// TwinCAT 3 PLC project ForgeExample
// ProgramVersion: 3.1.4026.17
// libraries:
//   Tc2_Standard, * (Beckhoff Automation GmbH)
//   Tc2_System, * (Beckhoff Automation GmbH)
//   Tc3_JsonXml, * (Beckhoff Automation GmbH)
//   Tc3_Module, * (Beckhoff Automation GmbH)
//   [Twincat Open Library], * (Home)
//   VisuSymbols,3.5.10.0,System
// project tree:
//   DUTs/ ST_CameraStates.TcDUT (not stored)
//   GVLs/ Hardware_Mapping.TcGVL (not stored), Cognex_Mapping.TcGVL (not stored)
//   / PlcTask.TcTTO
//   POUs/ MAIN.TcPOU, _5000_PRG_Aborting.TcPOU (not stored), _1000_PRG_Homing.TcPOU, _3000_PRG_Running.TcPOU (not stored), _2000_PRG_Stopping.TcPOU (not stored), _4000_PRG_Pausing.TcPOU (not stored), _6000_PRG_Proceeding.TcPOU (not stored)
// real-time tasks:
//   TASK PlcTask: cycle T#10ms, priority 20, ADS port 350
//   TASK VISU_TASK: cycle T#200000us, priority 30, ADS port 351
//   TASK IO Task New: cycle T#1ms, priority 1, ADS port 301
// motion (NC):
//   TASK NC-Task 1 SAF: cycle T#2ms, priority 4, ADS port 501
//   TASK NC-Task 1 SVB: cycle T#10ms, priority 8, ADS port 511
//   AXIS Axis 1 (id 1)
//     OtherSettings: AllowMotionCmdToSlave=true
//     encoder EncType=4
//       EncPara: MaxCount=#x0000ffff
//         Inc: RefSoftSyncMask=#x0000ffff
//     drive DrvType=24
//       Analog: TorqueSetpointScale=10, ScaleFactorActTorque=0.1
//       TimeComp: TaskDelayCycles=1
//     controller CtrType=1
//       CtrPara: PriorControlFactor=1
//         Observer: BandWidth=20
//   AXIS Axis 2 (id 2)
//     OtherSettings: AllowMotionCmdToSlave=true
//     encoder EncType=4
//       EncPara: MaxCount=#x0000ffff
//         Inc: RefSoftSyncMask=#x0000ffff
//     drive DrvType=24
//       Analog: TorqueSetpointScale=10, ScaleFactorActTorque=0.1
//       TimeComp: TaskDelayCycles=1
//     controller CtrType=1
//       CtrPara: PriorControlFactor=1
//         Observer: BandWidth=20
// I/O:
//   DEVICE Device 1 (TC3 EIP Scanner), AmsNetId 172.18.236.100.2.1
//     Box 1 (In-Sight 7000 Series) // <INFO> </INFO> <EDS> C:\TwinCAT\3.1\Config\Io\EtherNetIP\02A6006401090C00.eds </EDS>
//   DEVICE Device 2 (EtherCAT), AmsNetId 172.18.236.100.3.1
//     Term 2 (EK1100) [EK1100 EtherCAT Coupler (2A E-Bus)]
//       Term 3 (EL1008) [EL1008 8Ch. Dig. Input 24V, 3ms]
//       Term 4 (EL1008) [EL1008 8Ch. Dig. Input 24V, 3ms]
//       Term 5 (EL2008) [EL2008 8Ch. Dig. Output 24V, 0.5A]
//       Term 6 (EL2008) [EL2008 8Ch. Dig. Output 24V, 0.5A]
//       Term 7 (EL7047) [EL7047 1Ch. Stepper motor output stage (50V, 5A)]
//       Term 8 (EL7047) [EL7047 1Ch. Stepper motor output stage (50V, 5A)]
//       Term 8 (EL9011) [EL9011 End Terminal]
// variable links:
//   NC-Task 1 SAF/Axes/Axis 1 <-> Device 2 (EtherCAT)/Term 2 (EK1100)/Term 7 (EL7047)
//     Drive/Inputs/In/nState1 @bit 3 <-> STM Status/Status/Error
//     Drive/Inputs/In/nState1 @bit 7 <-> STM Status/Status/Motor stall
//     Drive/Inputs/In/nState1 @bit 5 <-> STM Status/Status/Moving negative
//     Drive/Inputs/In/nState1 @bit 4 <-> STM Status/Status/Moving positive
//     Drive/Inputs/In/nState1 @bit 1 <-> STM Status/Status/Ready
//     Drive/Inputs/In/nState1 <-> STM Status/Status/Ready to enable
//     Drive/Inputs/In/nState1 @bit 6 <-> STM Status/Status/Torque reduced
//     Drive/Inputs/In/nState1 @bit 2 <-> STM Status/Status/Warning
//     Drive/Inputs/In/nState2 @bit 3 <-> STM Status/Status/Digital input 1
//     Drive/Inputs/In/nState2 @bit 4 <-> STM Status/Status/Digital input 2
//     Drive/Inputs/In/nState2 @bit 5 <-> STM Status/Status/Sync error
//     Drive/Inputs/In/nState2 @bit 7 <-> STM Status/Status/TxPDO Toggle
//     Drive/Inputs/In/nState4 @bit 1 <-> WcState/InputToggle
//     Drive/Inputs/In/nState4 <-> WcState/WcState
//     Drive/Outputs/Out/nCtrl1 <-> STM Control/Control/Enable
//     Drive/Outputs/Out/nCtrl1 @bit 2 <-> STM Control/Control/Reduce torque
//     Drive/Outputs/Out/nCtrl1 @bit 1 <-> STM Control/Control/Reset
//     Drive/Outputs/Out/nCtrl2 @bit 3 <-> STM Control/Control/Digital output 1
//     Drive/Outputs/Out/nDataOut2[0] <-> STM Velocity/Velocity
//     Enc/Inputs/In/nDataIn1[0] <-> ENC Status compact/Counter value
//     Enc/Inputs/In/nDataIn2[0] <-> ENC Status compact/Latch value
//     Enc/Inputs/In/nState1 @bit 4 <-> ENC Status compact/Status/Counter overflow
//     Enc/Inputs/In/nState1 @bit 3 <-> ENC Status compact/Status/Counter underflow
//     Enc/Inputs/In/nState1 @bit 7 <-> ENC Status compact/Status/Extrapolation stall
//     Enc/Inputs/In/nState1 <-> ENC Status compact/Status/Latch C valid
//     Enc/Inputs/In/nState1 @bit 1 <-> ENC Status compact/Status/Latch extern valid
//     Enc/Inputs/In/nState1 @bit 2 <-> ENC Status compact/Status/Set counter done
//     Enc/Inputs/In/nState2 @bit 4 <-> ENC Status compact/Status/Status of extern latch
//     Enc/Inputs/In/nState2 <-> ENC Status compact/Status/Status of input A
//     Enc/Inputs/In/nState2 @bit 1 <-> ENC Status compact/Status/Status of input B
//     Enc/Inputs/In/nState2 @bit 2 <-> ENC Status compact/Status/Status of input C
//     Enc/Inputs/In/nState2 @bit 5 <-> ENC Status compact/Status/Sync error
//     Enc/Inputs/In/nState2 @bit 7 <-> ENC Status compact/Status/TxPDO Toggle
//     Enc/Inputs/In/nState4 @bit 1 <-> WcState/InputToggle
//     Enc/Inputs/In/nState4 <-> WcState/WcState
//     Enc/Outputs/Out/nCtrl1 <-> ENC Control compact/Control/Enable latch C
//     Enc/Outputs/Out/nCtrl1 @bit 3 <-> ENC Control compact/Control/Enable latch extern on negative edge
//     Enc/Outputs/Out/nCtrl1 @bit 1 <-> ENC Control compact/Control/Enable latch extern on positive edge
//     Enc/Outputs/Out/nCtrl1 @bit 2 <-> ENC Control compact/Control/Set counter
//     Enc/Outputs/Out/nDataOut1[0] <-> ENC Control compact/Set counter value
//   NC-Task 1 SAF/Axes/Axis 2 <-> Device 2 (EtherCAT)/Term 2 (EK1100)/Term 8 (EL7047)
//     Drive/Inputs/In/nState1 @bit 3 <-> STM Status/Status/Error
//     Drive/Inputs/In/nState1 @bit 7 <-> STM Status/Status/Motor stall
//     Drive/Inputs/In/nState1 @bit 5 <-> STM Status/Status/Moving negative
//     Drive/Inputs/In/nState1 @bit 4 <-> STM Status/Status/Moving positive
//     Drive/Inputs/In/nState1 @bit 1 <-> STM Status/Status/Ready
//     Drive/Inputs/In/nState1 <-> STM Status/Status/Ready to enable
//     Drive/Inputs/In/nState1 @bit 6 <-> STM Status/Status/Torque reduced
//     Drive/Inputs/In/nState1 @bit 2 <-> STM Status/Status/Warning
//     Drive/Inputs/In/nState2 @bit 3 <-> STM Status/Status/Digital input 1
//     Drive/Inputs/In/nState2 @bit 4 <-> STM Status/Status/Digital input 2
//     Drive/Inputs/In/nState2 @bit 5 <-> STM Status/Status/Sync error
//     Drive/Inputs/In/nState2 @bit 7 <-> STM Status/Status/TxPDO Toggle
//     Drive/Inputs/In/nState4 @bit 1 <-> WcState/InputToggle
//     Drive/Inputs/In/nState4 <-> WcState/WcState
//     Drive/Outputs/Out/nCtrl1 <-> STM Control/Control/Enable
//     Drive/Outputs/Out/nCtrl1 @bit 2 <-> STM Control/Control/Reduce torque
//     Drive/Outputs/Out/nCtrl1 @bit 1 <-> STM Control/Control/Reset
//     Drive/Outputs/Out/nCtrl2 @bit 3 <-> STM Control/Control/Digital output 1
//     Drive/Outputs/Out/nDataOut2[0] <-> STM Velocity/Velocity
//     Enc/Inputs/In/nDataIn1[0] <-> ENC Status compact/Counter value
//     Enc/Inputs/In/nDataIn2[0] <-> ENC Status compact/Latch value
//     Enc/Inputs/In/nState1 @bit 4 <-> ENC Status compact/Status/Counter overflow
//     Enc/Inputs/In/nState1 @bit 3 <-> ENC Status compact/Status/Counter underflow
//     Enc/Inputs/In/nState1 @bit 7 <-> ENC Status compact/Status/Extrapolation stall
//     Enc/Inputs/In/nState1 <-> ENC Status compact/Status/Latch C valid
//     Enc/Inputs/In/nState1 @bit 1 <-> ENC Status compact/Status/Latch extern valid
//     Enc/Inputs/In/nState1 @bit 2 <-> ENC Status compact/Status/Set counter done
//     Enc/Inputs/In/nState2 @bit 4 <-> ENC Status compact/Status/Status of extern latch
//     Enc/Inputs/In/nState2 <-> ENC Status compact/Status/Status of input A
//     Enc/Inputs/In/nState2 @bit 1 <-> ENC Status compact/Status/Status of input B
//     Enc/Inputs/In/nState2 @bit 2 <-> ENC Status compact/Status/Status of input C
//     Enc/Inputs/In/nState2 @bit 5 <-> ENC Status compact/Status/Sync error
//     Enc/Inputs/In/nState2 @bit 7 <-> ENC Status compact/Status/TxPDO Toggle
//     Enc/Inputs/In/nState4 @bit 1 <-> WcState/InputToggle
//     Enc/Inputs/In/nState4 <-> WcState/WcState
//     Enc/Outputs/Out/nCtrl1 <-> ENC Control compact/Control/Enable latch C
//     Enc/Outputs/Out/nCtrl1 @bit 3 <-> ENC Control compact/Control/Enable latch extern on negative edge
//     Enc/Outputs/Out/nCtrl1 @bit 1 <-> ENC Control compact/Control/Enable latch extern on positive edge
//     Enc/Outputs/Out/nCtrl1 @bit 2 <-> ENC Control compact/Control/Set counter
//     Enc/Outputs/Out/nDataOut1[0] <-> ENC Control compact/Set counter value
//   ForgeExample/ForgeExample Instance <-> Device 1 (TC3 EIP Scanner)/Box 1 (In-Sight 7000 Series)
//     PlcTask Inputs/Cognex_Mapping.inpAcquiring <-> Connection 1 (Input/Output)/Inputs/Acquiring
//     PlcTask Inputs/Cognex_Mapping.inpAcquisitionID <-> Connection 1 (Input/Output)/Inputs/Acquisition ID
//     PlcTask Inputs/Cognex_Mapping.inpCommandComplete <-> Connection 1 (Input/Output)/Inputs/Command Complete
//     PlcTask Inputs/Cognex_Mapping.inpCommandExecuting <-> Connection 1 (Input/Output)/Inputs/Command Executing
//     PlcTask Inputs/Cognex_Mapping.inpCommandFailed <-> Connection 1 (Input/Output)/Inputs/Command Failed
//     PlcTask Inputs/Cognex_Mapping.inpCurrentJobID <-> Connection 1 (Input/Output)/Inputs/Current Job ID
//     PlcTask Inputs/Cognex_Mapping.inpExposureComplete <-> Connection 1 (Input/Output)/Inputs/Exposure Complete
//     PlcTask Inputs/Cognex_Mapping.inpInspecting <-> Connection 1 (Input/Output)/Inputs/Inspecting
//     PlcTask Inputs/Cognex_Mapping.inpInspectionComplete <-> Connection 1 (Input/Output)/Inputs/Inspection Complete
//     PlcTask Inputs/Cognex_Mapping.inpInspectionID <-> Connection 1 (Input/Output)/Inputs/Inspection ID
//     PlcTask Inputs/Cognex_Mapping.inpInspectionResultCode <-> Connection 1 (Input/Output)/Inputs/Inspection Result Code
//     PlcTask Inputs/Cognex_Mapping.inpInspectionResults <-> Connection 1 (Input/Output)/Inputs/Inspection Results
//     PlcTask Inputs/Cognex_Mapping.inpJobPass <-> Connection 1 (Input/Output)/Inputs/Job Pass
//     PlcTask Inputs/Cognex_Mapping.inpMissedAcq <-> Connection 1 (Input/Output)/Inputs/Missed Acq
//     PlcTask Inputs/Cognex_Mapping.inpOfflineReason <-> Connection 1 (Input/Output)/Inputs/Offline Reason
//     PlcTask Inputs/Cognex_Mapping.inpOnline <-> Connection 1 (Input/Output)/Inputs/Online
//     PlcTask Inputs/Cognex_Mapping.inpResultsBufferOverrun <-> Connection 1 (Input/Output)/Inputs/Results Buffer Overrun
//     PlcTask Inputs/Cognex_Mapping.inpResultsValid <-> Connection 1 (Input/Output)/Inputs/Results Valid
//     PlcTask Inputs/Cognex_Mapping.inpTestRunReady <-> Connection 1 (Input/Output)/Inputs/Test Run Ready
//     PlcTask Inputs/Cognex_Mapping.inpTriggerAck <-> Connection 1 (Input/Output)/Inputs/Trigger Ack
//     PlcTask Inputs/Cognex_Mapping.inpTriggerReady <-> Connection 1 (Input/Output)/Inputs/Trigger Ready
//     PlcTask Outputs/Cognex_Mapping.outBufferResultsEnable <-> Connection 1 (Input/Output)/Outputs/Buffer Results Enable
//     PlcTask Outputs/Cognex_Mapping.outCommand <-> Connection 1 (Input/Output)/Outputs/Command
//     PlcTask Outputs/Cognex_Mapping.outExecuteCommand <-> Connection 1 (Input/Output)/Outputs/Execute Command
//     PlcTask Outputs/Cognex_Mapping.outInspectionResultsAck <-> Connection 1 (Input/Output)/Outputs/Inspection Results Ack
//     PlcTask Outputs/Cognex_Mapping.outSetOffline <-> Connection 1 (Input/Output)/Outputs/Set Offline
//     PlcTask Outputs/Cognex_Mapping.outSoftEvent{0..7} <-> Connection 1 (Input/Output)/Outputs/Soft Event {0..7}  (8 links)
//     PlcTask Outputs/Cognex_Mapping.outTriggerCamera <-> Connection 1 (Input/Output)/Outputs/Trigger
//     PlcTask Outputs/Cognex_Mapping.outTriggerEnable <-> Connection 1 (Input/Output)/Outputs/Trigger Enable
//     PlcTask Outputs/Cognex_Mapping.outUserData <-> Connection 1 (Input/Output)/Outputs/User Data
//   ForgeExample/ForgeExample Instance <-> Device 2 (EtherCAT)/Term 2 (EK1100)/Term 3 (EL1008)
//     PlcTask Inputs/Cognex_Mapping.input1 <-> Channel 1/Input
//     PlcTask Inputs/Cognex_Mapping.input2 <-> Channel 2/Input
//   ForgeExample/ForgeExample Instance <-> Device 2 (EtherCAT)/Term 2 (EK1100)/Term 5 (EL2008)
//     PlcTask Outputs/Cognex_Mapping.output1 <-> Channel 1/Output
//     PlcTask Outputs/Cognex_Mapping.output2 <-> Channel 2/Output

CONFIGURATION ForgeExample
    RESOURCE PLC ON TwinCAT3
        TASK PlcTask(INTERVAL := T#10ms, PRIORITY := 20);
        PROGRAM MAIN WITH PlcTask : MAIN;
    END_RESOURCE
END_CONFIGURATION

// ---- POUs/MAIN.TcPOU
PROGRAM MAIN
VAR
    fbStateMachine : FB_StateMachine;
    
    // Online-view command buttons — set TRUE in watch/online to trigger, auto-reset each scan
    btnHome    : BOOL;
    btnStart   : BOOL;
    btnStop    : BOOL;
    btnAbort   : BOOL;
    btnPause   : BOOL;
    btnProceed : BOOL;
    btnRetry   : BOOL;
	
	bTestcfgAutoRun : BOOL := TRUE;
END_VAR

fbStateMachine(
    EnableIn := TRUE,
    cfgAutoRun := bTestcfgAutoRun  // disable auto-run so manual buttons stay in control
);

// --- Online command buttons (write TRUE in TwinCAT online view to trigger) ---
IF btnHome    THEN fbStateMachine.Home();    btnHome    := FALSE; END_IF;
IF btnStart   THEN fbStateMachine.Start();   btnStart   := FALSE; END_IF;
IF btnStop    THEN fbStateMachine.Stop();    btnStop    := FALSE; END_IF;
IF btnAbort   THEN fbStateMachine.Abort();   btnAbort   := FALSE; END_IF;
IF btnPause   THEN fbStateMachine.Pause();   btnPause   := FALSE; END_IF;
IF btnProceed THEN fbStateMachine.Proceed(); btnProceed := FALSE; END_IF;
IF btnRetry   THEN fbStateMachine.Retry();   btnRetry   := FALSE; END_IF;

_1000_PRG_Homing(sm := fbStateMachine);
_3000_PRG_Running(sm := fbStateMachine);
_2000_PRG_Stopping(sm := fbStateMachine);
_5000_PRG_Aborting(sm := fbStateMachine);
_4000_PRG_Pausing(sm := fbStateMachine);
_6000_PRG_Proceeding(sm := fbStateMachine);

END_PROGRAM

// ---- POUs/_1000_PRG_Homing.TcPOU
PROGRAM _1000_PRG_Homing
VAR_IN_OUT
    sm : FB_StateMachine;
END_VAR
VAR
    step1000 : FB_Step;
    step1002 : FB_Step;
    step1004 : FB_Step;

    // Simulated hardware signals
    bDriveEnabled      : BOOL;
    bHomeSensorReached : BOOL;
    bServoReady        : BOOL;
    nRetryCount        : INT;
    tonHomeDelay       : TON;
END_VAR


//=============================================================================
// STEP 1000 - Initialize Homing
// Demonstrates: Entry (one-shot initialization), Execute (wait for perms),
//               Exiting (cleanup before advancing)
//=============================================================================
step1000(sm := sm, nStep := 1000, nNextStep := 1002, nTimeout := 10, sName := 'Init Homing');

IF step1000.Entry THEN
    // One-shot: reset state from any prior attempt
    bDriveEnabled := FALSE;
    bHomeSensorReached := FALSE;
    nRetryCount := 0;
    tonHomeDelay(IN := FALSE);  // reset timer
END_IF;

IF step1000.Execute THEN
    // Simulate: enable drive after a short delay
    tonHomeDelay(IN := TRUE, PT := T#2S);
    bDriveEnabled := tonHomeDelay.Q;

    // Permissives gate the transition to next step
    step1000.MapPerm(nIndex := 0, sDescription := 'Drive Enabled',      bValue := bDriveEnabled);
    step1000.MapPerm(nIndex := 1, sDescription := 'Safety Circuit OK',  bValue := TRUE);
    step1000.MapPerm(nIndex := 2, sDescription := 'No Active Faults',   bValue := TRUE);
END_IF;

IF step1000.Exiting THEN
    // One-shot cleanup: latch that initialization is done
    tonHomeDelay(IN := FALSE);
END_IF;

//=============================================================================
// STEP 1002 - Execute Homing Move
// Demonstrates: Entry (command actuator), Execute (monitor completion),
//               SetNextStep (dynamic branching on success/failure)
//=============================================================================
step1002(sm := sm, nStep := 1002, nNextStep := 1004, nTimeout := 20, sName := 'Execute Home Move');

IF step1002.Entry THEN
    // One-shot: command the axis to home
    bHomeSensorReached := FALSE;
    bServoReady := FALSE;
END_IF;

IF step1002.Execute THEN
    // Simulate homing motion completing after some time
    bHomeSensorReached := sm.Status.Step.TimerSeconds >= 5.0;
    bServoReady := bHomeSensorReached;

    step1002.MapPerm(nIndex := 0, sDescription := 'Home Sensor Reached', bValue := bHomeSensorReached);
    step1002.MapPerm(nIndex := 1, sDescription := 'Servo Settled',       bValue := bServoReady);
END_IF;

IF step1002.Exiting THEN
    // Could log completion or capture final position here
    ;
END_IF;

//=============================================================================
// STEP 1004 - Verify Home Position
// Demonstrates: Simple verification step, nNextStep := 0 ends the sequence
//=============================================================================
step1004(sm := sm, nStep := 1004, nNextStep := 0, nTimeout := 5, sName := 'Verify Home Position');

IF step1004.Entry THEN
    // Nothing special to initialize
    ;
END_IF;

IF step1004.Execute THEN
    // Verify the home position is stable
    step1004.MapPerm(nIndex := 0, sDescription := 'Position Stable', bValue := sm.Status.Step.TimerSeconds >= 1.0);
    step1004.MapPerm(nIndex := 1, sDescription := 'Encoder Valid',   bValue := TRUE);
END_IF;

END_PROGRAM
